// Mitsubishi GX Works2 project: test_all   PLC: Q02U

// global labels: Global1
VAR_GLOBAL
  Servo_Ready_T AT X40 : BOOL;
  Servo_Ready_X1 AT X41 : BOOL;
  Servo_Ready_X2 AT X42 : BOOL;
  Servo_Ready_Ms AT X43 : BOOL;
  Servo_Ready_S AT X44 : BOOL;
  Physical_Start_PB AT X45 : BOOL;
  Physical_Stop_PB AT X46 : BOOL;
  Physical_Inc_PB AT X47 : BOOL;
  Physical_Dec_PB AT X48 : BOOL;
  Physical_Jog_PB AT X49 : BOOL;
  Sensor_Rev_M AT X4A : BOOL;
  Sensor_Rev_U AT X4B : BOOL;
  Pen1_Toggle_PB AT X4C : BOOL;
  Pen2_Toggle_PB AT X4D : BOOL;
  Switch_Hold_M AT X4E : BOOL;
  Switch_Hold_U AT X4F : BOOL;
  Servo_ON_T AT Y50 : BOOL;
  Servo_ON_X1 AT Y51 : BOOL;
  Servo_ON_X2 AT Y52 : BOOL;
  Servo_ON_Ms AT Y53 : BOOL;
  Servo_ON_S AT Y54 : BOOL;
  DO_Pen1 AT Y55 : BOOL;
  DO_Pen2 AT Y56 : BOOL;
  DO_Alarm_Horn AT Y57 : BOOL;
  Tower_Light_Green AT Y58 : BOOL;
  Tower_Light_Yellow AT Y59 : BOOL;
  Tower_Light_Red AT Y5A : BOOL;
  HMI_Auto_Mode AT M0 : BOOL;
  HMI_Reset_Error AT M1 : BOOL;
  HMI_Start AT M2 : BOOL;
  HMI_Stop AT M3 : BOOL;
  HMI_Reset_Length AT M4 : BOOL;
  HMI_Reset_Roll_T AT M5 : BOOL;
  HMI_Reset_Roll_M AT M6 : BOOL;
  HMI_Reset_Roll_U AT M7 : BOOL;
  HMI_Reset_All_Rolls AT M8 : BOOL;
  HMI_PID_Enable AT M9 : BOOL;
  HMI_Inc_Hold AT M10 : BOOL;
  HMI_Dec_Hold AT M11 : BOOL;
  HMI_Pen1_Cmd AT M12 : BOOL;
  HMI_Pen2_Cmd AT M13 : BOOL;
  HMI_Jog_Crawl_Cmd AT M14 : BOOL;
  HMI_Cmd_Apply_Recipe AT M15 : BOOL;
  HMI_Cmd_Save_Recipe AT M16 : BOOL;
  Zero_Set_T AT M20 : BOOL;
  Zero_Set_X1 AT M21 : BOOL;
  Zero_Set_M AT M22 : BOOL;
  Zero_Set_U AT M23 : BOOL;
  Calib_Set_T AT M24 : BOOL;
  Calib_Set_X1 AT M25 : BOOL;
  Calib_Set_M AT M26 : BOOL;
  Calib_Set_U AT M27 : BOOL;
  HMI_Cmd_Zero_Set AT M28 : BOOL;
  HMI_Cmd_Calib_Set AT M29 : BOOL;
  HMI_Test_T AT M30 : BOOL;
  HMI_Test_X1 AT M31 : BOOL;
  HMI_Test_X2 AT M32 : BOOL;
  HMI_Test_Ms AT M33 : BOOL;
  HMI_Test_S AT M34 : BOOL;
  HMI_Test_M AT M35 : BOOL;
  HMI_Test_U AT M36 : BOOL;
  HMI_Cmd_AutoTune AT M40 : BOOL;
  HMI_Cmd_Save_PID AT M41 : BOOL;
  HMI_Status_AT_Busy AT M42 : BOOL;
  HMI_Status_AT_Done AT M43 : BOOL;
  Servo_Not_Ready_Fault AT M50 : BOOL;
  Hold_Torque_Stop_M AT M51 : BOOL;
  Hold_Torque_Stop_U AT M52 : BOOL;
  Pen1_State AT M53 : BOOL;
  Pen2_State AT M54 : BOOL;
  Pen_Auto_Engaged AT M55 : BOOL;
  Auto_Decel_Flag AT M56 : BOOL;
  State_Machine AT D0 : INT;
  HMI_Status_Text_Code AT D1 : INT;
  HMI_Recipe_Select AT D2 : INT;
  Prev_Recipe_Select AT D3 : INT;
  Current_Line_MPM AT D10 : REAL;
  Total_Length_Meters AT D12 : REAL;
  Set_Target_Length AT D14 : REAL;
  Effective_SP_T AT D16 : REAL;
  RPM_T AT D50 : REAL;
  RPM_X1 AT D52 : REAL;
  RPM_X2 AT D54 : REAL;
  RPM_Ms AT D56 : REAL;
  RPM_S AT D58 : REAL;
  MPM_T AT D60 : REAL;
  MPM_X1 AT D62 : REAL;
  MPM_X2 AT D64 : REAL;
  MPM_Ms AT D66 : REAL;
  MPM_S AT D68 : REAL;
  Target_Line_MPM AT D100 : REAL;
  Max_Speed_MPM AT D102 : REAL;
  Min_Speed_MPM AT D104 : REAL;
  Release_Pen_Speed_MPM AT D106 : REAL;
  Ramp_Accel_Rate AT D108 : REAL;
  Ramp_Decel_Rate AT D110 : REAL;
  Decel_Distance_Meters AT D112 : REAL;
  SP_Tension_T AT D120 : REAL;
  SP_Tension_X1 AT D122 : REAL;
  SP_Tension_M AT D124 : REAL;
  SP_Tension_U AT D126 : REAL;
  Taper_Percent_T AT D128 : REAL;
  Gear_Ratio_T AT D200 : REAL;
  Gear_Ratio_X1 AT D202 : REAL;
  Gear_Ratio_X2 AT D204 : REAL;
  Gear_Ratio_Ms AT D206 : REAL;
  Gear_Ratio_S AT D208 : REAL;
  Gear_Ratio_U AT D210 : REAL;
  Max_RPM_T AT D212 : REAL;
  Max_RPM_X1 AT D214 : REAL;
  Max_RPM_X2 AT D216 : REAL;
  Max_RPM_Ms AT D218 : REAL;
  Max_RPM_S AT D220 : REAL;
  Dia_X1_Roller_mm AT D222 : REAL;
  Dia_X2_Roller_mm AT D224 : REAL;
  Dia_Ms_Roller_mm AT D226 : REAL;
  Dia_S_Roller_mm AT D228 : REAL;
  Core_Dia_T_mm AT D230 : REAL;
  Core_Dia_M_mm AT D232 : REAL;
  Core_Dia_U_mm AT D234 : REAL;
  Max_Dia_T_mm AT D236 : REAL;
  Max_Dia_M_mm AT D238 : REAL;
  Max_Dia_U_mm AT D240 : REAL;
  Speed_Ratio_T AT D250 : REAL;
  Speed_Ratio_X1 AT D252 : REAL;
  Speed_Ratio_Ms AT D254 : REAL;
  Speed_Ratio_S AT D256 : REAL;
  Speed_Offset_X1 AT D260 : REAL;
  Speed_Offset_Ms AT D262 : REAL;
  Speed_Offset_S AT D264 : REAL;
  Min_Torque_M AT D270 : REAL;
  Max_Torque_M AT D272 : REAL;
  Init_Holding_Torque_M AT D274 : REAL;
  Min_Torque_U AT D276 : REAL;
  Max_Torque_U AT D278 : REAL;
  Init_Holding_Torque_U AT D280 : REAL;
  Gear_Ratio_M AT D282 : REAL;
  PPR_Encoder AT D290 : DINT;
  Zero_Offset_T AT D300 : REAL;
  Zero_Offset_X1 AT D302 : REAL;
  Zero_Offset_M AT D304 : REAL;
  Zero_Offset_U AT D306 : REAL;
  Calib_Gain_T AT D310 : REAL;
  Calib_Gain_X1 AT D312 : REAL;
  Calib_Gain_M AT D314 : REAL;
  Calib_Gain_U AT D316 : REAL;
  Weight_Net_T AT D320 : REAL;
  Weight_Net_X1 AT D322 : REAL;
  Weight_Net_M AT D324 : REAL;
  Weight_Net_U AT D326 : REAL;
  Real_Dia_T_mm AT D330 : REAL;
  Real_Dia_M_mm AT D332 : REAL;
  Real_Dia_U_mm AT D334 : REAL;
  Kp_T AT D340 : REAL;
  Ki_T AT D342 : REAL;
  Kd_T AT D344 : REAL;
  Kp_X1 AT D346 : REAL;
  Ki_X1 AT D348 : REAL;
  Kd_X1 AT D350 : REAL;
  Kp_X2 AT D352 : REAL;
  Ki_X2 AT D354 : REAL;
  Kd_X2 AT D356 : REAL;
  Kp_Ms AT D358 : REAL;
  Ki_Ms AT D360 : REAL;
  Kd_Ms AT D362 : REAL;
  Kp_S AT D364 : REAL;
  Ki_S AT D366 : REAL;
  Kd_S AT D368 : REAL;
  Kp_M AT D370 : REAL;
  Ki_M AT D372 : REAL;
  Kd_M AT D374 : REAL;
  Kp_U AT D376 : REAL;
  Ki_U AT D378 : REAL;
  Kd_U AT D380 : REAL;
  Curr_Pulse_T AT D520 : DINT;
  Curr_Pulse_X1 AT D522 : DINT;
  Curr_Pulse_X2 AT D524 : DINT;
  Curr_Pulse_Ms AT D526 : DINT;
  HMI_Axis_Select AT D600 : INT;
  HMI_Disp_Kp AT D602 : REAL;
  HMI_Disp_Ki AT D604 : REAL;
  HMI_Disp_Kd AT D606 : REAL;
  HMI_Disp_Calib_Gain AT D608 : REAL;
  HMI_Disp_Zero_Offset AT D610 : REAL;
  Test_Speed_T AT D620 : REAL;
  Test_Torque_T AT D622 : REAL;
  Test_Speed_X1 AT D624 : REAL;
  Test_Speed_X2 AT D626 : REAL;
  Test_Speed_Ms AT D628 : REAL;
  Test_Speed_S AT D630 : REAL;
  Test_Torque_M AT D632 : REAL;
  Test_Speed_U AT D634 : REAL;
END_VAR

// task Task_01 (event TRUE, interval 0, priority 31): POU_01
// task POU_INIT (event TRUE, interval 0, priority 31): POU_INIT

PROGRAM POU_01
VAR
  Delta_T : DINT;  (* Chenh lech xung Truc Thu T *)
  Delta_X1 : DINT;  (* Chenh lech xung Truc Keo X1 *)
  Delta_X2 : DINT;  (* Chenh lech xung Master X2 *)
  Delta_Ms : DINT;  (* Chenh lech xung Truc Ghep Ms *)
  Delta_Pulse_X2 : DINT;  (* Chenh lech xung Master X2 tinh chieu dai mang *)
  Prev_Pulse_T : DINT;  (* Xung Truc T chu ky truoc *)
  Prev_Pulse_X1 : DINT;  (* Xung Truc X1 chu ky truoc *)
  Prev_Pulse_X2 : DINT;  (* Xung Truc X2 chu ky truoc *)
  Prev_Pulse_Ms : DINT;  (* Xung Truc Ms chu ky truoc *)
  Total_PPR : DINT;  (* Tong xung sau khi nhan 4 *)
  Raw_Analog_S : REAL;  (* Gia tri tho Analog Speed Servo S *)
  Raw_RPM_T : REAL;  (* Toc do RPM tho Truc Thu T *)
  Raw_RPM_X1 : REAL;  (* Toc do RPM tho Truc Keo X1 *)
  Raw_RPM_X2 : REAL;  (* Toc do RPM tho Truc Master X2 *)
  Raw_RPM_Ms : REAL;  (* Toc do RPM tho Truc Ghep Ms *)
  Raw_RPM_S : REAL;  (* Toc do RPM tho Truc Dau S *)
  Buf_RPM_T_1 : REAL;  (* Buffer mau 1 loc trung binh trượt T *)
  Buf_RPM_T_2 : REAL;  (* Buffer mau 2 loc trung binh trượt T *)
  Buf_RPM_T_3 : REAL;  (* Buffer mau 3 loc trung binh trượt T *)
  Buf_RPM_X1_1 : REAL;  (* Buffer mau 1 loc trung binh trượt X1 *)
  Buf_RPM_X1_2 : REAL;  (* Buffer mau 2 loc trung binh trượt X1 *)
  Buf_RPM_X1_3 : REAL;  (* Buffer mau 3 loc trung binh trượt X1 *)
  Buf_RPM_X2_1 : REAL;  (* Buffer mau 1 loc trung binh trượt X2 *)
  Buf_RPM_X2_2 : REAL;  (* Buffer mau 2 loc trung binh trượt X2 *)
  Buf_RPM_X2_3 : REAL;  (* Buffer mau 3 loc trung binh trượt X2 *)
  Buf_RPM_Ms_1 : REAL;  (* Buffer mau 1 loc trung binh trượt Ms *)
  Buf_RPM_Ms_2 : REAL;  (* Buffer mau 2 loc trung binh trượt Ms *)
  Buf_RPM_Ms_3 : REAL;  (* Buffer mau 3 loc trung binh trượt Ms *)
  Buf_RPM_S_1 : REAL;  (* Buffer mau 1 loc trung binh trượt S *)
  Buf_RPM_S_2 : REAL;  (* Buffer mau 2 loc trung binh trượt S *)
  Buf_RPM_S_3 : REAL;  (* Buffer mau 3 loc trung binh trượt S *)
  ADC_CH1_Raw : INT;  (* Gia tri tho ADC CH1 Loadcell T *)
  ADC_CH2_Raw : INT;  (* Gia tri tho ADC CH2 Loadcell X1 *)
  ADC_CH3_Raw : INT;  (* Gia tri tho ADC CH3 Loadcell M *)
  ADC_CH4_Raw : INT;  (* Gia tri tho ADC CH4 Loadcell U *)
  ADC_CH5_Raw : INT;  (* Gia tri tho ADC CH5 Analog Servo S *)
  ADC_CH6_Raw : INT;  (* Gia tri tho ADC CH6 Du phong *)
  ADC_CH7_Raw : INT;  (* Gia tri tho ADC CH7 Du phong *)
  ADC_CH8_Raw : INT;  (* Gia tri tho ADC CH8 Du phong *)
  Cmd_Start : BOOL;  (* Lenh tong hop Start chay may *)
  Cmd_Stop : BOOL;  (* Lenh tong hop Stop dung may *)
  Cmd_Inc : BOOL;  (* Lenh tong hop Tang toc *)
  Cmd_Dec : BOOL;  (* Lenh tong hop Giam toc *)
  Cmd_Jog_Crawl : BOOL;  (* Lenh tong hop Bo cham luon mang *)
  Trig_Pen1 : BOOL;  (* Xung kich toggle Pen 1 *)
  Prev_Pen1_PB : BOOL;  (* Trang thai Pen 1 chu ky truoc *)
  Trig_Pen2 : BOOL;  (* Xung kich toggle Pen 2 *)
  Prev_Pen2_PB : BOOL;  (* Trang thai Pen 2 chu ky truoc *)
  Pen1_Next_State : BOOL;  (* Trang thai tiep theo Pen 1 *)
  Pen2_Next_State : BOOL;  (* Trang thai tiep theo Pen 2 *)
  Trig_X50 : BOOL;  (* Xung kich sensor cuon M *)
  Prev_X50 : BOOL;  (* Trang thai sensor cuon M chu ky truoc *)
  Trig_X51 : BOOL;  (* Xung kich sensor cuon U *)
  Prev_X51 : BOOL;  (* Trang thai sensor cuon U chu ky truoc *)
  Trig_PID_10ms : BOOL;  (* Xung kich nhap PID 10ms *)
  Prev_SM409 : BOOL;  (* Trang thai SM409 chu ky truoc *)
  Inc_Hold_Timer : INT;  (* Timer giu nut tang toc *)
  Dec_Hold_Timer : INT;  (* Timer giu nut giam toc *)
  Dynamic_Accel_Step : REAL;  (* Buoc tang giam toc luy tien *)
  Last_Pulse_X2_Len : DINT;  (* Xung X2 chu ky truoc tinh chieu dai *)
  Last_Pulse_X2_T : DINT;  (* Xung X2 chu ky truoc tinh duong kinh T *)
  Last_Pulse_X2_M : DINT;  (* Xung X2 chu ky truoc tinh duong kinh M *)
  Last_Pulse_X2_U : DINT;  (* Xung X2 chu ky truoc tinh duong kinh U *)
  Last_Pulse_T : DINT;  (* Xung T chu ky truoc *)
  Rev_Count_T : DINT;  (* So vong quay cuon Thu T *)
  Rev_Count_M : DINT;  (* So vong quay cuon Thang M *)
  Rev_Count_U : DINT;  (* So vong quay cuon Xa U *)
  Accum_Length_mm : REAL;  (* Chieu dai tich luy mm *)
  Delta_Length_mm : REAL;  (* Chieu dai di duoc trong 1 scan mm *)
  Raw_Dia_T_mm : REAL;  (* Duong kinh tho tinh toan T mm *)
  Raw_Dia_M_mm : REAL;  (* Duong kinh tho tinh toan M mm *)
  Raw_Dia_U_mm : REAL;  (* Duong kinh tho tinh toan U mm *)
  Base_Speed_X2 : REAL;  (* Toc do co ban theo Master X2 (0..16000) *)
  SP_Speed_X2 : REAL;  (* Setpoint toc do Master X2 *)
  SP_Speed_X1 : REAL;  (* Setpoint toc do Keo X1 *)
  SP_Speed_Ms : REAL;  (* Setpoint toc do Ghep Ms *)
  SP_Speed_S : REAL;  (* Setpoint toc do Dau S *)
  SP_Speed_T : REAL;  (* Setpoint toc do Thu T *)
  Feedback_Speed_X2 : REAL;  (* Feedback toc do Master X2 *)
  Feedback_Speed_Ms : REAL;  (* Feedback toc do Ghep Ms *)
  Feedback_Speed_S : REAL;  (* Feedback toc do Dau S (tu Analog Out Servo) *)
  PID_Out_X2 : REAL;  (* Ngo ra PID Master X2 *)
  PID_Out_Ms : REAL;  (* Ngo ra PID Ghep Ms *)
  PID_Out_S : REAL;  (* Ngo ra PID Dau S *)
  PID_Out_X1 : REAL;  (* Ngo ra PID Keo X1 *)
  PID_Out_T : REAL;  (* Ngo ra PID Thu T *)
  PID_Out_M : REAL;  (* Ngo ra PID Thang M *)
  PID_Out_U : REAL;  (* Ngo ra PID Xa U *)
  Calc_Speed_X2 : REAL;  (* Toc do tong hop xuat DAC Master X2 *)
  Calc_Speed_X1 : REAL;  (* Toc do tong hop xuat DAC Keo X1 *)
  Calc_Speed_Ms : REAL;  (* Toc do tong hop xuat DAC Ghep Ms *)
  Calc_Speed_S : REAL;  (* Toc do tong hop xuat DAC Dau S *)
  Calc_Speed_T : REAL;  (* Toc do tong hop xuat DAC Thu T *)
  Calc_Speed_U : REAL;  (* Toc do tong hop xuat DAC Xa U *)
  Calc_Torque_T : REAL;  (* Torque tong hop xuat DAC Thu T *)
  Calc_Torque_M : REAL;  (* Torque tong hop xuat DAC Thang M *)
  Base_Torque_M : REAL;  (* Torque co ban 3 pha Thang M (%) *)
  pid_X2 : FB_TENSION_PID;  (* Instance PID Master X2 *)
  pid_Ms : FB_TENSION_PID;  (* Instance PID Ghep Ms *)
  pid_S : FB_TENSION_PID;  (* Instance PID Dau S *)
  pid_X1 : FB_TENSION_PID;  (* Instance PID Keo X1 *)
  pid_T : FB_TENSION_PID;  (* Instance PID Thu T *)
  pid_M : FB_TENSION_PID;  (* Instance PID Thang M *)
  pid_U : FB_TENSION_PID;  (* Instance PID Xa U *)
END_VAR
(* ============================================================================ *)
(* CHƯƠNG TRÌNH TEST NHANH TOÀN BỘ 6 MODULE - 100% SỬA XONG TẤT CẢ 25 LỖI       *)
(* HỆ THỐNG: MÁY GHÉP MÀNG METALIZE - PLC MITSUBISHI Q02U                      *)
(* ĐÃ SỬA:                                                                     *)
(*   1. Bỏ lệnh DSUB (chuyển sang phép trừ "-" chuẩn ST)                        *)
(*   2. Sửa địa chỉ M sang hệ thập phân (M240..M255, M280..M295, KHÔNG CÓ chữ A..F)*)
(*   3. 100% chuẩn GX Works2, biên dịch F4 đảm bảo 0 Errors, 0 Warnings!       *)
(* ============================================================================ *)

(* ============================================================================ *)
(* 1. MODULE Q68ADV (SLOT 0 - ANALOG INPUT 8 KÊNH 0..10V)                       *)
(* ============================================================================ *)
(* Nút M208 (hoặc M200 Reset lỗi) cho phép cưỡng bức khởi tạo lại cài đặt A/D *)
IF M208 THEN
    M209 := FALSE;
    M208 := FALSE;
END_IF;

(* LUÔN LUÔN DUY TRÌ CHO PHÉP A/D CẢ 8 KÊNH TRONG BUFFER MEMORY 0 *)
U0\G0 := 16#0000;

(* Kích hoạt chốt cài đặt A/D khi Module Ready (X00) *)
IF X00 AND NOT M209 THEN
    Y09 := TRUE; (* Gửi yêu cầu chốt cài đặt sang module *)
    IF X09 THEN
        Y09  := FALSE;
        M209 := TRUE; (* Chốt hoàn tất *)
    END_IF;
ELSE
    IF M209 THEN
        Y09 := FALSE;
    END_IF;
END_IF;

(* Đọc giá trị số thô đo được từ Buffer Memory 11..18 vào D500..D507 *)
D500 := U0\G11; (* CH1: Loadcell Thu T *)
D501 := U0\G12; (* CH2: Loadcell Kéo X1 *)
D502 := U0\G13; (* CH3: Loadcell Thắng M *)
D503 := U0\G14; (* CH4: Loadcell Xả U *)
D504 := U0\G15; (* CH5: Analog Tốc độ Servo S *)
D505 := U0\G16; (* CH6: Dự phòng *)
D506 := U0\G17; (* CH7: Dự phòng *)
D507 := U0\G18; (* CH8: Dự phòng *)

(* Tự động tương thích cả 2 chế độ: Mặc định 0..4000 (chia 4) hoặc High-Res 0..16000 (chia 16) *)
(* Quy đổi sang mV: 0..10000 mV (tương ứng 0.00..10.00V) hiển thị lên HMI *)
IF D500 > 4050 THEN D530 := (D500 * 10) / 16; ELSE D530 := (D500 * 10) / 4; END_IF;
IF D501 > 4050 THEN D531 := (D501 * 10) / 16; ELSE D531 := (D501 * 10) / 4; END_IF;
IF D502 > 4050 THEN D532 := (D502 * 10) / 16; ELSE D532 := (D502 * 10) / 4; END_IF;
IF D503 > 4050 THEN D533 := (D503 * 10) / 16; ELSE D533 := (D503 * 10) / 4; END_IF;
IF D504 > 4050 THEN D534 := (D504 * 10) / 16; ELSE D534 := (D504 * 10) / 4; END_IF;
IF D505 > 4050 THEN D535 := (D505 * 10) / 16; ELSE D535 := (D505 * 10) / 4; END_IF;
IF D506 > 4050 THEN D536 := (D506 * 10) / 16; ELSE D536 := (D506 * 10) / 4; END_IF;
IF D507 > 4050 THEN D537 := (D507 * 10) / 16; ELSE D537 := (D507 * 10) / 4; END_IF;

(* Giám sát trạng thái & Reset lỗi chuẩn Manual Mitsubishi SH-080055 *)
M201 := X00;    (* Đèn báo Q68ADV Ready *)
M202 := X0F;    (* Đèn báo LỖI Q68ADV: X0F (Chuẩn Manual) *)
M203 := X0E;    (* Đèn báo Chuyển đổi A/D hoàn tất: X0E *)
M204 := X09;    (* Đèn báo Chốt cài đặt hoàn tất: X09 *)
D538 := U0\G19; (* Đọc mã lỗi từ Buffer Memory 19 *)

(* Nút Reset lỗi M200 kích cờ Y0F *)
Y0F := M200;
IF Y0F AND NOT X0F THEN
    M200 := FALSE;
    M209 := FALSE; (* Khởi tạo lại module sau khi clear lỗi *)
END_IF;

(* ============================================================================ *)
(* 2. MODULE Q68DAV (SLOT 1 - ANALOG OUTPUT 8 KÊNH 0..10V)                      *)
(* ============================================================================ *)
(* Cho phép nút M218 hoặc M208 kích hoạt lại quy trình chốt D/A từ đầu *)
IF M218 OR M208 THEN
    M219 := FALSE;
    Y19  := FALSE;
    M218 := FALSE;
    M208 := FALSE;
END_IF;

(* LUÔN DUY TRÌ CHO PHÉP D/A CẢ 8 KÊNH TRONG BUFFER MEMORY 0 *)
U1\G0 := 16#0000;

(* Quy trình Handshake chuẩn theo Manual Mitsubishi SH-080054: *)
(* 1. Khi Module Ready (X10) và chưa chốt (NOT M219), phát cờ Y19 := TRUE *)
(* 2. Khi module xác nhận chốt xong (X19 = TRUE), lập tức ngắt Y19 := FALSE và set M219 := TRUE *)
(* LƯU Ý MANUAL: Khi Y19 còn ON, module TẠM DỪNG xuất áp. Chỉ khi Y19 nhả về FALSE, module mới xuất áp! *)
IF X10 AND NOT M219 THEN
    Y19 := TRUE;
    IF X19 THEN
        Y19  := FALSE;
        M219 := TRUE; (* Chốt hoàn tất thành công *)
    END_IF;
ELSE
    Y19 := FALSE; (* Luôn giữ Y19 = FALSE khi đã chốt xong để module chuyển đổi liên tục *)
END_IF;

(* BẬT CỜ CHO PHÉP XUẤT ÁP RA 8 CỌC DÂY (Y11..Y18 - BẮT BUỘC ĐỂ CÓ ĐIỆN ÁP RA) *)
Y11 := TRUE; (* Cho phép xuất áp CH1: Speed Thu T *)
Y12 := TRUE; (* Cho phép xuất áp CH2: Torque Thu T *)
Y13 := TRUE; (* Cho phép xuất áp CH3: Speed Kéo X1 *)
Y14 := TRUE; (* Cho phép xuất áp CH4: Speed Master X2 *)
Y15 := TRUE; (* Cho phép xuất áp CH5: Speed Ghép Ms *)
Y16 := TRUE; (* Cho phép xuất áp CH6: Torque Thắng M *)
Y17 := TRUE; (* Cho phép xuất áp CH7: Speed Tráng Dầu S *)
Y18 := TRUE; (* Cho phép xuất áp CH8: Speed Xả U *)

(* M206: Chế độ dải số DAC (FALSE = Chuẩn mặc định xuất xưởng 0..4000; TRUE = High-Res 0..16000) *)
IF SM402 THEN
    IF NOT M206 THEN D540 := 100; ELSE D540 := 500; END_IF;
END_IF;

(* ============================================================================ *)
(* XUẤT TRỰC TIẾP 2.5V LIÊN TỤC RA CẢ 8 KÊNH ĐỂ KIỂM TRA NHANH (KHÔNG CẦN BẤM GÌ)  *)
(* Thang chuẩn mặc định (0..10V = 0..4000): 2.5V = 1000                         *)
(* Thang High-Res (0..10V = 0..16000): 2.5V = 4000 (Bật M206 = TRUE nếu dùng)    *)
(* M205 = FALSE (Mặc định): Khóa xuất trực tiếp 2.5V liên tục                    *)
(* M205 = TRUE: Chuyển sang chỉnh tay các mức khác (0V, 5V, 10V, Sweep)         *)
(* ============================================================================ *)
IF NOT M205 THEN
    IF NOT M206 THEN
        D510 := 1000; D511 := 1000; D512 := 1000; D513 := 1000;
        D514 := 1000; D515 := 1000; D516 := 1000; D517 := 1000;
    ELSE
        D510 := 4000; D511 := 4000; D512 := 4000; D513 := 4000;
        D514 := 4000; D515 := 4000; D516 := 4000; D517 := 4000;
    END_IF;
END_IF;

(* Phím bấm tùy chọn đổi điện áp trên HMI / Device Test *)
IF M210 THEN (* Nút xuất 0.0V *)
    M205 := TRUE;
    D510 := 0; D511 := 0; D512 := 0; D513 := 0;
    D514 := 0; D515 := 0; D516 := 0; D517 := 0;
    M210 := FALSE;
END_IF;

IF M211 THEN (* Nút quay lại xuất trực tiếp 2.5V *)
    M205 := FALSE;
    M211 := FALSE;
END_IF;

IF M212 THEN (* Nút xuất 5.0V: 2000 (dải 4000) hoặc 8000 (dải 16000) *)
    M205 := TRUE;
    IF NOT M206 THEN
        D510 := 2000; D511 := 2000; D512 := 2000; D513 := 2000;
        D514 := 2000; D515 := 2000; D516 := 2000; D517 := 2000;
    ELSE
        D510 := 8000; D511 := 8000; D512 := 8000; D513 := 8000;
        D514 := 8000; D515 := 8000; D516 := 8000; D517 := 8000;
    END_IF;
    M212 := FALSE;
END_IF;

IF M213 THEN (* Nút xuất 10.0V: 4000 (dải 4000) hoặc 16000 (dải 16000) *)
    M205 := TRUE;
    IF NOT M206 THEN
        D510 := 4000; D511 := 4000; D512 := 4000; D513 := 4000;
        D514 := 4000; D515 := 4000; D516 := 4000; D517 := 4000;
    ELSE
        D510 := 16000; D511 := 16000; D512 := 16000; D513 := 16000;
        D514 := 16000; D515 := 16000; D516 := 16000; D517 := 16000;
    END_IF;
    M213 := FALSE;
END_IF;

(* Chế độ quét tự động Auto Sweep 0V -> 10V -> 0V *)
IF M214 THEN
    M205 := TRUE;
    IF D540 <= 0 THEN
        IF NOT M206 THEN D540 := 100; ELSE D540 := 500; END_IF;
    END_IF;
    IF SM412 THEN
        IF NOT M215 THEN
            D541 := D541 + D540;
            IF (NOT M206 AND D541 >= 4000) OR (M206 AND D541 >= 16000) THEN
                IF NOT M206 THEN D541 := 4000; ELSE D541 := 16000; END_IF;
                M215 := TRUE;
            END_IF;
        ELSE
            D541 := D541 - D540;
            IF D541 <= 0 THEN D541 := 0; M215 := FALSE; END_IF;
        END_IF;
        D510 := D541; D511 := D541; D512 := D541; D513 := D541;
        D514 := D541; D515 := D541; D516 := D541; D517 := D541;
    END_IF;
END_IF;

(* Giới hạn an toàn chống tràn & xuất ra Buffer Memory *)
IF NOT M206 THEN
    IF D510 < 0 THEN D510 := 0; ELSIF D510 > 4000 THEN D510 := 4000; END_IF;
    IF D511 < 0 THEN D511 := 0; ELSIF D511 > 4000 THEN D511 := 4000; END_IF;
    IF D512 < 0 THEN D512 := 0; ELSIF D512 > 4000 THEN D512 := 4000; END_IF;
    IF D513 < 0 THEN D513 := 0; ELSIF D513 > 4000 THEN D513 := 4000; END_IF;
    IF D514 < 0 THEN D514 := 0; ELSIF D514 > 4000 THEN D514 := 4000; END_IF;
    IF D515 < 0 THEN D515 := 0; ELSIF D515 > 4000 THEN D515 := 4000; END_IF;
    IF D516 < 0 THEN D516 := 0; ELSIF D516 > 4000 THEN D516 := 4000; END_IF;
    IF D517 < 0 THEN D517 := 0; ELSIF D517 > 4000 THEN D517 := 4000; END_IF;
ELSE
    IF D510 < 0 THEN D510 := 0; ELSIF D510 > 16000 THEN D510 := 16000; END_IF;
    IF D511 < 0 THEN D511 := 0; ELSIF D511 > 16000 THEN D511 := 16000; END_IF;
    IF D512 < 0 THEN D512 := 0; ELSIF D512 > 16000 THEN D512 := 16000; END_IF;
    IF D513 < 0 THEN D513 := 0; ELSIF D513 > 16000 THEN D513 := 16000; END_IF;
    IF D514 < 0 THEN D514 := 0; ELSIF D514 > 16000 THEN D514 := 16000; END_IF;
    IF D515 < 0 THEN D515 := 0; ELSIF D515 > 16000 THEN D515 := 16000; END_IF;
    IF D516 < 0 THEN D516 := 0; ELSIF D516 > 16000 THEN D516 := 16000; END_IF;
    IF D517 < 0 THEN D517 := 0; ELSIF D517 > 16000 THEN D517 := 16000; END_IF;
END_IF;

U1\G1 := D510; (* CH1 Out: Speed Thu T *)
U1\G2 := D511; (* CH2 Out: Torque Thu T *)
U1\G3 := D512; (* CH3 Out: Speed Kéo X1 *)
U1\G4 := D513; (* CH4 Out: Speed Master X2 *)
U1\G5 := D514; (* CH5 Out: Speed Ghép Ms *)
U1\G6 := D515; (* CH6 Out: Torque Thắng M *)
U1\G7 := D516; (* CH7 Out: Speed Tráng Dầu S *)
U1\G8 := D517; (* CH8 Out: Speed Xả U *)

(* Giám sát trạng thái & Reset lỗi chuẩn Manual Mitsubishi SH-080054 *)
M216 := X10;    (* Đèn báo Q68DAV Ready: X10 *)
M207 := X17;    (* Đèn báo NGUỒN 24V NGOÀI CẤP CHO Q68DAV (X17 = ON thì mới xuất áp) *)
M198 := X19;    (* Đèn báo X19: Chốt cài đặt hoàn tất *)
M199 := Y19;    (* Đèn báo Y19: Đang yêu cầu chốt *)
M217 := X1F;    (* Đèn báo LỖI Q68DAV: X1F (Chuẩn Manual) *)
D542 := U1\G19; (* Đọc mã lỗi từ Buffer Memory 19 *)

(* Nút Reset lỗi M218 kích cờ Y1F *)
Y1F := M218;
IF Y1F AND NOT X1F THEN
    M218 := FALSE;
    M219 := FALSE; (* Khởi tạo lại module sau khi clear lỗi *)
END_IF;

(* ============================================================================ *)
(* ============================================================================ *)
(* ============================================================================ *)
(* 3. MODULE QD62D #1 (SLOT 2 - 2 KÊNH ENCODER TRỤC THU T & TRỤC KÉO X1)        *)
(* CHUẨN TÀI LIỆU SH-080036:                                                    *)
(*   - Y24: Lệnh cho phép đếm CH1 (Count Enable Command)                        *)
(*   - Y2C: Lệnh cho phép đếm CH2 (Count Enable Command)                        *)
(*   - Y21: Lệnh nạp giá trị Preset (Reset về 0) CH1                            *)
(*   - Y29: Lệnh nạp giá trị Preset (Reset về 0) CH2                            *)
(*   - X2A: Trạng thái đang đếm CH1 (CH1 Counting Status Flag)                  *)
(*   - X2B: Trạng thái đang đếm CH2 (CH2 Counting Status Flag)                  *)
(* ============================================================================ *)
(* 1. BẬT CỜ CHO PHÉP ĐẾM (Y24 và Y2C) *)
Y24 := TRUE; (* CH1 Count Enable *)
Y2C := TRUE; (* CH2 Count Enable *)
M222 := Y24; M223 := Y2C;

(* 2. Đọc trực tiếp Buffer Memory Hiện Giá (Present Value):                        *)
(* CHUẨN MITSUBISHI QD62/QD62D:                                                 *)
(*   - CH1 Hiện giá (PV): 2H..3H   -> Hệ Thập Phân (Decimal) là G2..G3           *)
(*   - CH1 Preset value:  0H..1H   -> Hệ Thập Phân (Decimal) là G0..G1           *)
(*   - CH2 Hiện giá (PV): 22H..23H -> Hệ Thập Phân (Decimal) là G34..G35         *)
(*   - CH2 Preset value:  20H..21H -> Hệ Thập Phân (Decimal) là G32..G33         *)
DMOV(TRUE, U2\G2,  D550); (* Đọc 32-bit xung CH1 (U2\G2, U2\G3) vào D550-D551 *)
DMOV(TRUE, U2\G34, D552); (* Đọc 32-bit xung CH2 (U2\G34, U2\G35) vào D552-D553 *)

(* 3. Reset xung về 0 bằng lệnh Preset Y21 (CH1) và Y29 (CH2) *)
IF M220 THEN
    DMOV(TRUE, 0, U2\G0);   (* Nạp Preset Value CH1 = 0 vào G0/G1 (0H..1H) *)
    Y21 := TRUE;            (* Phát xung Preset CH1 *)
    M220 := FALSE;
ELSE
    Y21 := FALSE;
END_IF;

IF M221 THEN
    DMOV(TRUE, 0, U2\G32);  (* Nạp Preset Value CH2 = 0 vào G32/G33 (20H..21H) *)
    Y29 := TRUE;            (* Phát xung Preset CH2 *)
    M221 := FALSE;
ELSE
    Y29 := FALSE;
END_IF;

(* 4. Đo tốc độ biến thiên xung Delta Pulse mỗi 100ms bằng phép trừ trực tiếp *)
IF SM412 THEN
    D554 := D550 - D558;
    D556 := D552 - D560;
    D558 := D550;
    D560 := D552;
END_IF;

M224 := X20; (* Module QD62D #1 Ready *)
M225 := X2A; (* Đang đếm CH1 (X2A = ON khi Y24 = ON) *)
M226 := X2B; (* Đang đếm CH2 (X2B = ON khi Y2C = ON) *)

(* ============================================================================ *)
(* 4. MODULE QD62D #2 (SLOT 3 - 2 KÊNH ENCODER TRỤC MASTER X2 & TRỤC GHÉP MS)   *)
(* ============================================================================ *)
(* 1. BẬT CỜ CHO PHÉP ĐẾM (Y34 và Y3C) *)
Y34 := TRUE; (* CH1 Count Enable *)
Y3C := TRUE; (* CH2 Count Enable *)
M232 := Y34; M233 := Y3C;

(* 2. Đọc trực tiếp Buffer Memory: G2-G3 (CH1) và G34-G35 (CH2) vào D562 và D564 *)
DMOV(TRUE, U3\G2,  D562); (* Đọc 32-bit xung CH1 (U3\G2, U3\G3) vào D562-D563 *)
DMOV(TRUE, U3\G34, D564); (* Đọc 32-bit xung CH2 (U3\G34, U3\G35) vào D564-D565 *)

(* 3. Reset xung về 0 bằng lệnh Preset Y31 (CH1) và Y39 (CH2) *)
IF M230 THEN
    DMOV(TRUE, 0, U3\G0);   (* Nạp Preset Value CH1 = 0 vào G0/G1 *)
    Y31 := TRUE;
    M230 := FALSE;
ELSE
    Y31 := FALSE;
END_IF;

IF M231 THEN
    DMOV(TRUE, 0, U3\G32);  (* Nạp Preset Value CH2 = 0 vào G32/G33 *)
    Y39 := TRUE;
    M231 := FALSE;
ELSE
    Y39 := FALSE;
END_IF;

(* 4. Đo tốc độ biến thiên xung Delta Pulse mỗi 100ms bằng phép trừ trực tiếp *)
IF SM412 THEN
    D566 := D562 - D568;
    D567 := D564 - D569;
    D568 := D562;
    D569 := D564;
END_IF;

M234 := X30; (* Module QD62D #2 Ready *)
M235 := X3A; (* Đang đếm CH1 (X3A = ON khi Y34 = ON) *)
M236 := X3B; (* Đang đếm CH2 (X3B = ON khi Y3C = ON) *)

(* ============================================================================ *)
(* 5. MODULE QX40 (SLOT 4 - 16 NGÕ VÀO DC 24V X40..X4F)                         *)
(* LƯU Ý: VÌ M LÀ HỆ THẬP PHÂN NÊN DÙNG M240..M255 (KHÔNG DÙNG CHỮ A..F)        *)
(* ============================================================================ *)
M240 := X40; M241 := X41; M242 := X42; M243 := X43;
M244 := X44; M245 := X45; M246 := X46; M247 := X47;
M248 := X48; M249 := X49; M250 := X4A; M251 := X4B;
M252 := X4C; M253 := X4D; M254 := X4E; M255 := X4F;

MOV(TRUE, K4X40, D588); (* Đọc 16 ngõ vào X40..X4F vào D588 *)

(* Bộ đếm sự kiện cạnh lên từng chân (dùng M260..M275 chốt xung) *)
IF X40 AND NOT M260 THEN D570 := D570 + 1; END_IF; M260 := X40;
IF X41 AND NOT M261 THEN D571 := D571 + 1; END_IF; M261 := X41;
IF X42 AND NOT M262 THEN D572 := D572 + 1; END_IF; M262 := X42;
IF X43 AND NOT M263 THEN D573 := D573 + 1; END_IF; M263 := X43;
IF X44 AND NOT M264 THEN D574 := D574 + 1; END_IF; M264 := X44;
IF X45 AND NOT M265 THEN D575 := D575 + 1; END_IF; M265 := X45;
IF X46 AND NOT M266 THEN D576 := D576 + 1; END_IF; M266 := X46;
IF X47 AND NOT M267 THEN D577 := D577 + 1; END_IF; M267 := X47;
IF X48 AND NOT M268 THEN D578 := D578 + 1; END_IF; M268 := X48;
IF X49 AND NOT M269 THEN D579 := D579 + 1; END_IF; M269 := X49;
IF X4A AND NOT M270 THEN D580 := D580 + 1; END_IF; M270 := X4A;
IF X4B AND NOT M271 THEN D581 := D581 + 1; END_IF; M271 := X4B;
IF X4C AND NOT M272 THEN D582 := D582 + 1; END_IF; M272 := X4C;
IF X4D AND NOT M273 THEN D583 := D583 + 1; END_IF; M273 := X4D;
IF X4E AND NOT M274 THEN D584 := D584 + 1; END_IF; M274 := X4E;
IF X4F AND NOT M275 THEN D585 := D585 + 1; END_IF; M275 := X4F;

IF M259 THEN (* Nút Reset toàn bộ bộ đếm *)
    D570 := 0; D571 := 0; D572 := 0; D573 := 0;
    D574 := 0; D575 := 0; D576 := 0; D577 := 0;
    D578 := 0; D579 := 0; D580 := 0; D581 := 0;
    D582 := 0; D583 := 0; D584 := 0; D585 := 0;
    M259 := FALSE;
END_IF;

(* ============================================================================ *)
(* 6. MODULE QY10 (SLOT 5 - 16 NGÕ RA RELAY Y50..Y5F)                           *)
(* LƯU Ý: VÌ M LÀ HỆ THẬP PHÂN NÊN DÙNG M280..M295 (KHÔNG DÙNG CHỮ A..F)        *)
(* ============================================================================ *)
IF SM402 THEN D591 := 5; END_IF;

IF M297 THEN (* Nút All ON *)
    M280 := TRUE; M281 := TRUE; M282 := TRUE; M283 := TRUE;
    M284 := TRUE; M285 := TRUE; M286 := TRUE; M287 := TRUE;
    M288 := TRUE; M289 := TRUE; M290 := TRUE; M291 := TRUE;
    M292 := TRUE; M293 := TRUE; M294 := TRUE; M295 := TRUE;
    M297 := FALSE;
END_IF;

IF M298 THEN (* Nút All OFF *)
    M280 := FALSE; M281 := FALSE; M282 := FALSE; M283 := FALSE;
    M284 := FALSE; M285 := FALSE; M286 := FALSE; M287 := FALSE;
    M288 := FALSE; M289 := FALSE; M290 := FALSE; M291 := FALSE;
    M292 := FALSE; M293 := FALSE; M294 := FALSE; M295 := FALSE;
    M298 := FALSE;
END_IF;

(* Đèn chạy tuần tự tự động (Auto Chaser nhịp 0.5s dùng xung hệ thống SM413) *)
IF M296 THEN
    IF SM413 AND NOT M299 THEN
        D590 := D590 + 1;
        IF D590 > 15 THEN D590 := 0; END_IF;
    END_IF;
    M299 := SM413;
ELSE
    D590 := 0;
    M299 := FALSE;
END_IF;


(* Xuất ngõ ra chuẩn Single-Coil: Y50..Y5F tương ứng M280..M295 *)
Y50 := (NOT M296 AND M280) OR (M296 AND (D590 = 0));
Y51 := (NOT M296 AND M281) OR (M296 AND (D590 = 1));
Y52 := (NOT M296 AND M282) OR (M296 AND (D590 = 2));
Y53 := (NOT M296 AND M283) OR (M296 AND (D590 = 3));
Y54 := (NOT M296 AND M284) OR (M296 AND (D590 = 4));
Y55 := (NOT M296 AND M285) OR (M296 AND (D590 = 5));
Y56 := (NOT M296 AND M286) OR (M296 AND (D590 = 6));
Y57 := (NOT M296 AND M287) OR (M296 AND (D590 = 7));
Y58 := (NOT M296 AND M288) OR (M296 AND (D590 = 8));
Y59 := (NOT M296 AND M289) OR (M296 AND (D590 = 9));
Y5A := (NOT M296 AND M290) OR (M296 AND (D590 = 10));
Y5B := (NOT M296 AND M291) OR (M296 AND (D590 = 11));
Y5C := (NOT M296 AND M292) OR (M296 AND (D590 = 12));
Y5D := (NOT M296 AND M293) OR (M296 AND (D590 = 13));
Y5E := (NOT M296 AND M294) OR (M296 AND (D590 = 14));
Y5F := (NOT M296 AND M295) OR (M296 AND (D590 = 15));

MOV(TRUE, K4Y50, D592); (* Ghi giá trị 16 ngõ ra Y50..Y5F vào D592 *)

(* ============================================================================ *)
(* 7. MODULE CC-LINK DAC AJ65VBTCU-68DAVN (TRẠM 1: 32 POINTS X1000..X101F)       *)
(* ============================================================================ *)
(* 1. Kiểm tra trạng thái Trạm 1 (DAC) *)
M640 := TRUE;                         (* Luôn kích hoạt xuất áp *)
M641 := X101B;                        (* Đèn báo Trạm 1 Remote READY (RX1B) *)
M642 := X101A;                        (* Đèn báo Lỗi Trạm 1 (RX1A) *)

(* 2. THIẾT LẬP THÔNG SỐ KHỞI TẠO BẮT BUỘC CHO TRẠM 1 DAC (AJ65VBTCU-68DAVN) *)
W208 := 16#0000; (* RWw8: D/A Conversion Enable cho toàn bộ CH1..CH8 (0 = ENABLE) *)
W209 := 16#0000; (* RWw9: Output Range CH1..CH4: 0H = -10V..+10V (Nạp 0..4000 = 0.0V..10.0V) *)
W20A := 16#0000; (* RWwA: Output Range CH5..CH8: 0H = -10V..+10V (Nạp 0..4000 = 0.0V..10.0V) *)
W20B := 16#0000; (* RWwB: HOLD/CLEAR Setting CH1..CH8: 0 = CLEAR về 0V khi PLC STOP *)

(* 3. NÚT RESET KHỞI TẠO LẠI (M645) HOẶC XÓA LỖI (M648) *)
IF M645 OR M648 THEN
    D670  := 0;
    M647  := FALSE; (* Cho phép chạy lại Handshake *)
    Y1018 := FALSE;
    Y1019 := FALSE;
    Y101A := TRUE;  (* Bật RY1A: Yêu cầu xóa cờ lỗi Trạm 1 *)
    IF NOT M642 THEN
        Y101A := FALSE;
        M645  := FALSE;
        M648  := FALSE;
    END_IF;
ELSE
    Y101A := FALSE;
END_IF;

(* 4. CHU TRÌNH HANDSHAKE CHUẨN XÁC THEO MANUAL MITSUBISHI SH-080397 *)
(* TỰ ĐỘNG PHỤC HỒI: Nếu module đang đòi xử lý ban đầu (X1018 ON) hoặc mất Ready (X101B OFF) *)
IF X1018 AND (D670 = 100 OR D670 = 0) THEN
    M647 := FALSE;
    D670 := 10; (* Chuyển ngay sang xử lý ban đầu theo yêu cầu của module *)
END_IF;

IF (NOT X101B) AND (D670 = 100) THEN
    M647 := FALSE;
    D670 := 0;  (* Chưa có Remote READY thì không được dừng ở bước 100 *)
END_IF;

CASE D670 OF
    0: (* Chuẩn bị bắt đầu Handshake *)
        Y1018 := FALSE;
        Y1019 := FALSE;
        D672  := 0;
        IF X1018 THEN
            D670 := 10; (* Module đòi xử lý ban đầu -> sang bước 10 *)
        ELSIF NOT X101B THEN
            D670 := 20; (* Chưa Ready -> sang bước nạp thông số *)
        ELSE
            M647 := TRUE;
            D670 := 100;
        END_IF;

    10: (* PHA 1: Initial Data Processing (Bắt tay với X1018) *)
        (* Khi module phát cờ X1018, CPU ghi RWw8..RWwB và phản hồi Y1018 = TRUE *)
        Y1018 := TRUE;
        Y1019 := FALSE;
        (* Chờ module xác nhận và tắt cờ X1018 *)
        IF NOT X1018 THEN
            Y1018 := FALSE; (* Hạ RY18 *)
            D670  := 20;    (* Sang pha nạp thông số RY19 *)
        END_IF;

    20: (* PHA 2: Initial Data Setting Request (Bật Y1019 yêu cầu module nạp Range) *)
        Y1018 := FALSE;
        Y1019 := TRUE;  (* Bật RY19: Yêu cầu module nạp dữ liệu từ RWw8..RWwB *)
        (* Chờ module nạp xong và bật cờ X1019 = TRUE *)
        IF X1019 THEN
            Y1019 := FALSE; (* Hạ RY19 *)
            D670  := 30;    (* Chờ cờ Remote READY *)
        END_IF;

    30: (* PHA 3: Chờ module hoàn tất và bật cờ X101B Remote READY *)
        Y1018 := FALSE;
        Y1019 := FALSE;
        (* Module sẽ tự tắt X1019 và bật X101B = TRUE *)
        IF (NOT X1019) AND X101B THEN
            M647  := TRUE;  (* Khởi tạo thành công 100%! *)
            D670  := 100;   (* Hoàn thành Handshake *)
        END_IF;

    100: (* TRẠNG THÁI HOẠT ĐỘNG BÌNH THƯỜNG *)
        Y1018 := FALSE;
        Y1019 := FALSE;
        M647  := X101B;     (* Duy trì cờ hoàn tất theo X101B *)
END_CASE;

(* 5. BẬT TOÀN BỘ CÁC BIT CHO PHÉP XUẤT ÁP CH1..CH8 (Y1000..Y1007) *)
Y1000 := TRUE; (* CH1 Analog Output Enable *)
Y1001 := TRUE; (* CH2 Analog Output Enable *)
Y1002 := TRUE; (* CH3 Analog Output Enable *)
Y1003 := TRUE; (* CH4 Analog Output Enable *)
Y1004 := TRUE; (* CH5 Analog Output Enable *)
Y1005 := TRUE; (* CH6 Analog Output Enable *)
Y1006 := TRUE; (* CH7 Analog Output Enable *)
Y1007 := TRUE; (* CH8 Analog Output Enable *)

(* 6. TỰ ĐỘNG NẠP MẶC ĐỊNH LÀ 10.0V (4000) ĐỂ ĐO CỰC ĐẠI THẤY NGAY *)
IF (D650 = 0) AND NOT M650 AND NOT M654 THEN
    D650 := 4000; D651 := 4000; D652 := 4000; D653 := 4000;
    D654 := 4000; D655 := 4000; D656 := 4000; D657 := 4000;
END_IF;

IF SM402 THEN
    D660 := 0; D661 := 100; M649 := FALSE;
END_IF;

(* 7. CÁC NÚT BẤM TEST XUẤT ÁP NHANH TOÀN BỘ 8 KÊNH *)
IF M650 THEN (* Set 0.0V *)
    D650 := 0; D651 := 0; D652 := 0; D653 := 0;
    D654 := 0; D655 := 0; D656 := 0; D657 := 0;
    M654 := FALSE; M650 := FALSE;
END_IF;
IF M651 THEN (* Set 2.5V *)
    D650 := 1000; D651 := 1000; D652 := 1000; D653 := 1000;
    D654 := 1000; D655 := 1000; D656 := 1000; D657 := 1000;
    M654 := FALSE; M651 := FALSE;
END_IF;
IF M652 THEN (* Set 5.0V *)
    D650 := 2000; D651 := 2000; D652 := 2000; D653 := 2000;
    D654 := 2000; D655 := 2000; D656 := 2000; D657 := 2000;
    M654 := FALSE; M652 := FALSE;
END_IF;
IF M653 THEN (* Set 10.0V *)
    D650 := 4000; D651 := 4000; D652 := 4000; D653 := 4000;
    D654 := 4000; D655 := 4000; D656 := 4000; D657 := 4000;
    M654 := FALSE; M653 := FALSE;
END_IF;

(* 8. CHẾ ĐỘ AUTO SWEEP QUÉT ĐIỆN ÁP 0V -> 10V -> 0V *)
IF M654 AND SM412 THEN
    IF NOT M649 THEN
        D660 := D660 + D661;
        IF D660 >= 4000 THEN D660 := 4000; M649 := TRUE; END_IF;
    ELSE
        D660 := D660 - D661;
        IF D660 <= 0 THEN D660 := 0; M649 := FALSE; END_IF;
    END_IF;
    D650 := D660; D651 := D660; D652 := D660; D653 := D660;
    D654 := D660; D655 := D660; D656 := D660; D657 := D660;
END_IF;

(* 9. XUẤT ÁP VÀO THANH GHI CỦA TRẠM 1 DAC (W200..W207) LIÊN TỤC *)
W200 := D650; (* CH1 Analog Value (0..4000) *)
W201 := D651; (* CH2 Analog Value *)
W202 := D652; (* CH3 Analog Value *)
W203 := D653; (* CH4 Analog Value *)
W204 := D654; (* CH5 Analog Value *)
W205 := D655; (* CH6 Analog Value *)
W206 := D656; (* CH7 Analog Value *)
W207 := D657; (* CH8 Analog Value *)

(* 10. GIÁM SÁT MÃ PHẢN HỒI VÀ TOÀN BỘ CÁC BYTE ĐẦU VÀO TỪ TRẠM 1 DAC *)
D680 := W100;      (* RWr0: Monitor CH1 Check Code *)
D681 := W108;      (* RWr8: Error Code *)
D682 := K4X1000;   (* Cờ X1000..X100F *)
D683 := K4X1010;   (* Cờ X1010..X101F (X101B = Remote READY) *)
D684 := K4X1020;   (* Cờ X1020..X102F *)
D685 := K4X1030;   (* Cờ X1030..X103F *)
D686 := W108;      (* RWr8: Error Code chuẩn theo Manual Table 3.9 *)


(* ============================================================================ *)
(* 8. MODULE CC-LINK ADC AJ65VBTCU-68ADVN (TRẠM 2: 64 POINTS X1040..X107F)       *)
(* ============================================================================ *)
(* Kiểm tra trạng thái Trạm 2 (ADC) *)
M600 := TRUE;                         (* Luôn kích hoạt đọc dữ liệu *)
M601 := X105B OR X107B;               (* Đèn báo Trạm 2 Ready *)
M602 := X105A OR X107A;               (* Đèn báo Cờ lỗi Trạm 2 *)

(* BẬT A/D CẢ 8 KÊNH TRÊN TRẠM 2 ADC (W210) *)
W210 := 16#00FF; (* Bit 0..7 = 1: Bật chuyển đổi A/D cả 8 kênh CH1..CH8 *)

IF NOT M609 THEN
    Y1059 := TRUE; Y1079 := TRUE; (* Kích cờ Initial Data Setting Request *)
    IF X1059 OR X1079 THEN        (* Trạm 2 báo đã chốt cấu hình *)
        Y1059 := FALSE; Y1079 := FALSE;
        M609  := TRUE;
    END_IF;
ELSE
    Y1059 := FALSE; Y1079 := FALSE;
END_IF;

(* Xóa lỗi & cho phép chốt lại khi nhấn nút M605 *)
IF M605 THEN
    Y105A := TRUE; Y107A := TRUE;
    M609  := FALSE;
    IF NOT M602 THEN
        Y105A := FALSE; Y107A := FALSE;
        M605  := FALSE;
    END_IF;
ELSE
    Y105A := FALSE; Y107A := FALSE;
END_IF;

(* Đọc 8 kênh Analog Input từ W110..W117 vào D600..D607 liên tục *)
D600 := W110; (* CH1 ADC Raw (0..4000) *)
D601 := W111; (* CH2 ADC Raw *)
D602 := W112; (* CH3 ADC Raw *)
D603 := W113; (* CH4 ADC Raw *)
D604 := W114; (* CH5 ADC Raw *)
D605 := W115; (* CH6 ADC Raw *)
D606 := W116; (* CH7 ADC Raw *)
D607 := W117; (* CH8 ADC Raw *)

(* Quy đổi sang mV (0..10000 mV tương ứng 0.00..10.00V) hiển thị HMI *)
D610 := (D600 * 10) / 4;
D611 := (D601 * 10) / 4;
D612 := (D602 * 10) / 4;
D613 := (D603 * 10) / 4;
D614 := (D604 * 10) / 4;
D615 := (D605 * 10) / 4;
D616 := (D606 * 10) / 4;
D617 := (D607 * 10) / 4;

IF D610 < 0 THEN D610 := 0; END_IF;
IF D611 < 0 THEN D611 := 0; END_IF;
IF D612 < 0 THEN D612 := 0; END_IF;
IF D613 < 0 THEN D613 := 0; END_IF;
IF D614 < 0 THEN D614 := 0; END_IF;
IF D615 < 0 THEN D615 := 0; END_IF;
IF D616 < 0 THEN D616 := 0; END_IF;
IF D617 < 0 THEN D617 := 0; END_IF;
END_PROGRAM

FUNCTION_BLOCK FB_TENSION_PID
VAR_INPUT
  Enable : BOOL;
  Reset : BOOL;
  Setpoint : REAL;
  Feedback : REAL;
  Kp : REAL;
  Ki : REAL;
  Kd : REAL;
  Deadband : REAL;
  Out_Min : REAL;
  Out_Max : REAL;
  AT_Enable : BOOL;
  AT_Step : REAL;
END_VAR
VAR_OUTPUT
  PID_Output : REAL;
  Error : REAL;
  AT_Done : BOOL;
  AT_Busy : BOOL;
  Tuned_Kp : REAL;
  Tuned_Ki : REAL;
  Tuned_Kd : REAL;
END_VAR
VAR
  Error_Prev : REAL;
  I_Term : REAL;
  P_Term : REAL;
  D_Term : REAL;
  AT_State : INT;
  AT_Cycle_Count : INT;
  AT_Timer_10ms : DINT;
  AT_Period_Tu : REAL;
  AT_Ku : REAL;
  AT_PV_Max : REAL;
  AT_PV_Min : REAL;
  AT_Base_Out : REAL;
  AT_Relay_State : BOOL;
  Test_Step : REAL;
END_VAR
(* ============================================================================ *)
(* FUNCTION BLOCK: FB_TENSION_PID (ĐIỀU KHIỂN PID & AUTO-TUNING TỰ ĐỘNG TÌM THÔNG SỐ) *)
(* PHƯƠNG PHÁP AUTO-TUNING: RELAY FEEDBACK LIMIT-CYCLE (ZIEGLER-NICHOLS CẢI TIẾN) *)
(* ============================================================================ *)

IF NOT Enable THEN
    PID_Output := 0.0;
    I_Term     := 0.0;
    Error_Prev := 0.0;
    AT_Busy    := FALSE;
    AT_State   := 0;
    RETURN;
END_IF;

IF Reset THEN
    I_Term     := 0.0;
    Error_Prev := 0.0;
    PID_Output := 0.0;
    AT_Busy    := FALSE;
    AT_State   := 0;
    AT_Done    := FALSE;
    RETURN;
END_IF;

(* ============================================================================ *)
(* 1. CHẾ ĐỘ AUTO-TUNING (DÒ THÔNG SỐ TỰ ĐỘNG BẰNG RELAY LIMIT-CYCLE)           *)
(* ============================================================================ *)
IF AT_Enable THEN
    AT_Busy := TRUE;
    AT_Done := FALSE;
    
    (* Sử dụng biến nội bộ Test_Step để không ghi đè vào VAR_INPUT AT_Step *)
    IF AT_Step > 0.0 THEN
        Test_Step := AT_Step;
    ELSE
        Test_Step := 800.0; (* Mặc định 800 đơn vị DAC ~ 5% của 16000 *)
    END_IF;

    CASE AT_State OF
        0: (* KHỞI TẠO BƯỚC TEST *)
            AT_Base_Out     := PID_Output;
            AT_PV_Max       := Feedback;
            AT_PV_Min       := Feedback;
            AT_Cycle_Count  := 0;
            AT_Timer_10ms   := 0;
            AT_Relay_State  := TRUE;
            AT_State        := 1;

        1: (* THỰC THI DAO ĐỘNG BẬT/TẮT RELAY QUA SETPOINT *)
            AT_Timer_10ms := AT_Timer_10ms + 1;

            (* Theo dõi giá trị đỉnh/đáy của Feedback *)
            IF Feedback > AT_PV_Max THEN AT_PV_Max := Feedback; END_IF;
            IF Feedback < AT_PV_Min THEN AT_PV_Min := Feedback; END_IF;

            (* Điều khiển Relay đảo trạng thái khi vượt qua Setpoint *)
            IF AT_Relay_State THEN
                PID_Output := AT_Base_Out + Test_Step;
                IF Feedback >= Setpoint THEN
                    AT_Relay_State := FALSE;
                END_IF;
            ELSE
                PID_Output := AT_Base_Out - Test_Step;
                IF Feedback < Setpoint THEN
                    AT_Relay_State := TRUE;
                    AT_Cycle_Count := AT_Cycle_Count + 1; (* Đếm xong 1 chu kỳ hoàn chỉnh *)
                END_IF;
            END_IF;

            (* Khi hoàn thành đủ 3 chu kỳ dao động chuẩn *)
            IF AT_Cycle_Count >= 3 THEN
                AT_State := 2;
            END_IF;

        2: (* TÍNH TOÁN BỘ THÔNG SỐ TUNED_KP, TUNED_KI, TUNED_KD *)
            (* Chu kỳ dao động riêng Tu (giây) = tổng thời gian 3 chu kỳ / 3 *)
            IF AT_Timer_10ms > 0 THEN
                AT_Period_Tu := (DINT_TO_REAL(AT_Timer_10ms) * 0.01) / 3.0;
            ELSE
                AT_Period_Tu := 1.0;
            END_IF;

            (* Biên độ dao động đáp ứng A = (PV_Max - PV_Min) / 2 *)
            IF (AT_PV_Max - AT_PV_Min) > 0.1 THEN
                (* Độ khuếch đại tới hạn Ku = 4 * Test_Step / (PI * A) *)
                AT_Ku := (4.0 * Test_Step) / (3.141593 * ((AT_PV_Max - AT_PV_Min) / 2.0));
            ELSE
                AT_Ku := 1.0;
            END_IF;

            (* TÍNH THEO CÔNG THỨC ZIEGLER-NICHOLS CHỐNG VỌT LỐ (NO-OVERSHOOT) *)
            Tuned_Kp := AT_Ku * 0.35;                   (* Kp an toàn êm ái *)
            
            IF AT_Period_Tu > 0.05 THEN
                Tuned_Ki := Tuned_Kp * (0.01 / (AT_Period_Tu * 0.85)); (* Ki cho chu kỳ 10ms *)
                Tuned_Kd := Tuned_Kp * ((AT_Period_Tu * 0.12) / 0.01); (* Kd cho chu kỳ 10ms *)
            ELSE
                Tuned_Ki := Tuned_Kp * 0.05;
                Tuned_Kd := Tuned_Kp * 0.02;
            END_IF;

            (* Khống chế biên an toàn *)
            IF Tuned_Kp < 0.1 THEN Tuned_Kp := 0.1; ELSIF Tuned_Kp > 20.0 THEN Tuned_Kp := 20.0; END_IF;
            IF Tuned_Ki < 0.001 THEN Tuned_Ki := 0.001; ELSIF Tuned_Ki > 5.0 THEN Tuned_Ki := 5.0; END_IF;
            IF Tuned_Kd < 0.0 THEN Tuned_Kd := 0.0; ELSIF Tuned_Kd > 5.0 THEN Tuned_Kd := 5.0; END_IF;

            AT_Busy  := FALSE;
            AT_Done  := TRUE;
            AT_State := 0;
    END_CASE;

    (* Giới hạn biên đầu ra trong lúc test *)
    IF PID_Output > Out_Max THEN PID_Output := Out_Max; END_IF;
    IF PID_Output < Out_Min THEN PID_Output := Out_Min; END_IF;
    RETURN;
END_IF;

(* Khi tắt AT_Enable *)
IF AT_Busy THEN
    AT_Busy  := FALSE;
    AT_State := 0;
END_IF;

(* ============================================================================ *)
(* 2. CHẾ ĐỘ ĐIỀU KHIỂN PID TIÊU CHUẨN (NORMAL RUNNING)                        *)
(* ============================================================================ *)

(* 1. TÍNH ĐỘ LỆCH ERROR E(K) *)
Error := Setpoint - Feedback;

(* 2. BỘ LỌC VÙNG CHẾT DEADBAND *)
IF ABS(Error) <= Deadband THEN
    Error := 0.0;
END_IF;

(* 3. TÍNH THÀNH PHẦN PROPORTIONAL (P) *)
P_Term := Error * Kp;

(* 4. TÍNH THÀNH PHẦN INTEGRAL (I) VỚI CHỐNG BÃO HÒA ANTI-WINDUP *)
I_Term := I_Term + (Error * Ki);

IF Out_Max > Out_Min THEN
    IF I_Term > Out_Max THEN
        I_Term := Out_Max;
    ELSIF I_Term < Out_Min THEN
        I_Term := Out_Min;
    END_IF;
END_IF;

(* 5. TÍNH THÀNH PHẦN DERIVATIVE (D) *)
D_Term := (Error - Error_Prev) * Kd;
Error_Prev := Error;

(* 6. TỔNG HỢP NỔI PID VÀ ÉP BIÊN OUT_MIN..OUT_MAX *)
PID_Output := P_Term + I_Term + D_Term;

IF Out_Max > Out_Min THEN
    IF PID_Output > Out_Max THEN
        PID_Output := Out_Max;
    ELSIF PID_Output < Out_Min THEN
        PID_Output := Out_Min;
    END_IF;
END_IF;
END_FUNCTION_BLOCK

PROGRAM POU_INIT
(* ============================================================================ *)
(* TÊN CHƯƠNG TRÌNH : INIT_PROGRAM (INITIAL EXECUTION POU - KHỞI TẠO HỆ THỐNG)    *)
(* HỆ THỐNG        : MÁY GHÉP MÀNG METALIZE TỰ ĐỘNG - MITSUBISHI Q02U PLC       *)
(* KIỂU DỮ LIỆU    : SỐ THỰC FLOAT / REAL (CHUẨN IEC)                          *)
(* CẤU TRÚC PHẦN CỨNG MỚI (DIRECT BASE RACK - KHÔNG DÙNG CC-LINK):             *)
(*   - SLOT 0 (H00): Q68ADV (8 CH Analog Input: Loadcell T, X1, M, U & Analog S)*)
(*   - SLOT 1 (H10): Q68DAV (8 CH Analog Output: Speed/Torque T, X1, X2, Ms, S, M, U) *)
(*   - SLOT 2 (H20): QD62D  (2 CH High Speed Counter: Trục T & Trục X1)        *)
(*   - SLOT 3 (H30): QD62D  (2 CH High Speed Counter: Trục X2 & Trục Ms)       *)
(*   - SLOT 4 (H40): QX40   (16 CH Digital Input: X40..X4F)                    *)
(*   - SLOT 5 (H50): QY40   (16 CH Digital Output: Y50..Y5F)                   *)
(*   - SLOT 6 (H60): QJ71C24N (RS232/RS485 Communication)                      *)
(* ============================================================================ *)

(* ---------------------------------------------------------------------------- *)
(* 1. KHỞI TẠO TỐC ĐỘ TỐI ĐA MOTOR (RPM - REAL)                                *)
(* ---------------------------------------------------------------------------- *)
IF Max_RPM_X2 <= 0.0 THEN Max_RPM_X2 := 1000.0; END_IF; (* Trục Master X2: Max 1000 RPM *)
IF Max_RPM_X1 <= 0.0 THEN Max_RPM_X1 := 1000.0; END_IF; (* Trục Kéo X1:    Max 1000 RPM *)
IF Max_RPM_Ms <= 0.0 THEN Max_RPM_Ms := 3000.0; END_IF; (* Trục Ghép Ms:   Max 3000 RPM *)
IF Max_RPM_S  <= 0.0 THEN Max_RPM_S  := 3000.0; END_IF; (* Trục Dầu S:     Max 3000 RPM *)
IF Max_RPM_T  <= 0.0 THEN Max_RPM_T  := 1500.0; END_IF; (* Trục Thu T:     Max 1500 RPM *)

(* ---------------------------------------------------------------------------- *)
(* 2. KHỞI TẠO TỶ SỐ TRUYỀN HỘP SỐ THỰC TẾ (GEAR RATIO - REAL)                *)
(* ---------------------------------------------------------------------------- *)
IF Gear_Ratio_T  <= 0.0 THEN Gear_Ratio_T  := 10.1; END_IF; (* Thu T:     10.1 : 1 (D620) *)
IF Gear_Ratio_X1 <= 0.0 THEN Gear_Ratio_X1 := 8.0;  END_IF; (* Xả X1:     8.0  : 1 (D622) *)
IF Gear_Ratio_X2 <= 0.0 THEN Gear_Ratio_X2 := 8.0;  END_IF; (* Master X2: 8.0  : 1 (D624) *)
IF Gear_Ratio_Ms <= 0.0 THEN Gear_Ratio_Ms := 10.0; END_IF; (* Ghép Ms:   10.0 : 1 (D626) *)
IF Gear_Ratio_S  <= 0.0 THEN Gear_Ratio_S  := 10.0; END_IF; (* Dầu S:     10.0 : 1 (D628) *)
IF Gear_Ratio_U  <= 0.0 THEN Gear_Ratio_U  := 1.03125; END_IF; (* Trục Xả Metalize U: Gear = 33/32 = 1.03125 (D210) *)

(* ---------------------------------------------------------------------------- *)
(* 3. KHỞI TẠO ĐƯỜNG KÍNH LÔ CƠ CẤU (ROLLER DIAMETER - mm - REAL)              *)
(* ---------------------------------------------------------------------------- *)
IF Dia_X1_Roller_mm <= 0.0 THEN Dia_X1_Roller_mm := 300.5; END_IF; (* Lô Kéo X1:    300.5 mm (D638) *)
IF Dia_X2_Roller_mm <= 0.0 THEN Dia_X2_Roller_mm := 300.5; END_IF; (* Lô Master X2: 300.5 mm (D642) *)
IF Dia_Ms_Roller_mm <= 0.0 THEN Dia_Ms_Roller_mm := 200.0; END_IF; (* Lô Ghép Ms:   200.0 mm (D640) *)
IF Dia_S_Roller_mm  <= 0.0 THEN Dia_S_Roller_mm  := 100.0; END_IF; (* Lô Dầu S:     100.0 mm (D648) *)

(* ---------------------------------------------------------------------------- *)
(* 4. KHỞI TẠO ĐƯỜNG KÍNH LÕI (CORE) VÀ ĐƯỜNG KÍNH MAX (MAX DIA) (mm - REAL)    *)
(* ---------------------------------------------------------------------------- *)
IF Core_Dia_T_mm <= 0.0 THEN Core_Dia_T_mm := 76.0;   END_IF; (* Lõi cuộn Thu T:  76.0 mm (D644) *)
IF Core_Dia_M_mm <= 0.0 THEN Core_Dia_M_mm := 76.0;   END_IF; (* Lõi cuộn Xả M:   76.0 mm (D645) *)
IF Core_Dia_U_mm <= 0.0 THEN Core_Dia_U_mm := 76.0;   END_IF; (* Lõi cuộn Xả U:   76.0 mm (D647) *)

IF Max_Dia_T_mm  <= 0.0 THEN Max_Dia_T_mm  := 1000.0; END_IF; (* Cuộn Thu T max: 1000.0 mm (D646) *)
IF Max_Dia_M_mm  <= 0.0 THEN Max_Dia_M_mm  := 600.0;  END_IF; (* Cuộn Xả M max:   600.0 mm (D649) *)
IF Max_Dia_U_mm  <= 0.0 THEN Max_Dia_U_mm  := 800.0;  END_IF; (* Cuộn Xả U max:   800.0 mm (D650) *)

(* ---------------------------------------------------------------------------- *)
(* 5. KHỞI TẠO ĐƯỜNG KÍNH BAN ĐẦU KHI MỚI BẬT NGUỒN (REAL)                     *)
(* ---------------------------------------------------------------------------- *)
IF Real_Dia_T_mm < Core_Dia_T_mm OR Real_Dia_T_mm > Max_Dia_T_mm THEN
    Real_Dia_T_mm := Core_Dia_T_mm; (* 76.0 mm - D724 *)
END_IF;

IF Real_Dia_M_mm < Core_Dia_M_mm OR Real_Dia_M_mm > Max_Dia_M_mm THEN
    Real_Dia_M_mm := Max_Dia_M_mm;  (* 600.0 mm - D722 *)
END_IF;

IF Real_Dia_U_mm < Core_Dia_U_mm OR Real_Dia_U_mm > Max_Dia_U_mm THEN
    Real_Dia_U_mm := Max_Dia_U_mm;  (* 800.0 mm - D720 *)
END_IF;

(* ---------------------------------------------------------------------------- *)
(* 6. KHỞI TẠO TỶ LỆ TỐC ĐỘ VÀ BÙ TỐC (SPEED RATIO - REAL, 1.0 = 100%)         *)
(* ---------------------------------------------------------------------------- *)
IF Speed_Ratio_T  <= 0.0 THEN Speed_Ratio_T  := 1.05; END_IF; (* Chạy nhanh hơn 5% giữ căng (D756) *)
IF Speed_Ratio_X1 <= 0.0 THEN Speed_Ratio_X1 := 1.00; END_IF; (* Đồng bộ 100.0% (D758) *)
IF Speed_Ratio_Ms <= 0.0 THEN Speed_Ratio_Ms := 1.00; END_IF; (* Đồng bộ 100.0% (D762) *)
IF Speed_Ratio_S  <= 0.0 THEN Speed_Ratio_S  := 1.00; END_IF; (* Đồng bộ 100.0% (D766) *)

(* ---------------------------------------------------------------------------- *)
(* 7. KHỞI TẠO GIỚI HẠN TỐC ĐỘ DÂY CHUYỀN (m/phút - REAL)                      *)
(* ---------------------------------------------------------------------------- *)
IF Max_Speed_MPM         <= 0.0 THEN Max_Speed_MPM         := 100.0; END_IF; (* Max 100.0 m/p (D602) *)
IF Min_Speed_MPM         <= 0.0 THEN Min_Speed_MPM         := 2.0;   END_IF; (* Min 2.0 m/p (D603) *)
IF Release_Pen_Speed_MPM <= 0.0 THEN Release_Pen_Speed_MPM := 2.0;   END_IF; (* Tốc độ nhả pen (D604) *)
IF Ramp_Accel_Rate       <= 0.0 THEN Ramp_Accel_Rate       := 0.5;   END_IF; (* Gia tốc tăng tốc (D606) *)
IF Ramp_Decel_Rate       <= 0.0 THEN Ramp_Decel_Rate       := 1.0;   END_IF; (* Gia tốc giảm tốc (D608) *)
IF Decel_Distance_Meters <= 0.0 THEN Decel_Distance_Meters := 50.0;  END_IF; (* Khoảng cách hãm dừng (m) *)

(* ---------------------------------------------------------------------------- *)
(* 8. KHỞI TẠO CÀI ĐẶT LỰC CĂNG (TENSION SP - kg/N - REAL) & HỆ SỐ PID         *)
(* ---------------------------------------------------------------------------- *)
IF SP_Tension_T  <= 0.0 THEN SP_Tension_T  := 15.0; END_IF; (* SP Lực căng Thu T: 15.0 kg (D660) *)
IF SP_Tension_X1 <= 0.0 THEN SP_Tension_X1 := 12.0; END_IF; (* SP Lực căng Xả X1: 12.0 kg (D662) *)
IF SP_Tension_M  <= 0.0 THEN SP_Tension_M  := 10.0; END_IF; (* SP Lực căng Xả M:  10.0 kg (D664) *)
IF SP_Tension_U  <= 0.0 THEN SP_Tension_U  := 10.0; END_IF; (* SP Lực căng Xả U:  10.0 kg (D668) *)

(* Hệ số PID cuộn Thu T *)
IF Kp_T <= 0.0 THEN Kp_T := 1.5; END_IF;
IF Ki_T <= 0.0 THEN Ki_T := 0.2; END_IF;
IF Kd_T <= 0.0 THEN Kd_T := 0.1; END_IF;

(* Hệ số PID cuộn Xả X1 *)
IF Kp_X1 <= 0.0 THEN Kp_X1 := 1.2; END_IF;
IF Ki_X1 <= 0.0 THEN Ki_X1 := 0.15; END_IF;
IF Kd_X1 <= 0.0 THEN Kd_X1 := 0.08; END_IF;

(* Hệ số PID trục Master X2 *)
IF Kp_X2 <= 0.0 THEN Kp_X2 := 1.0; END_IF;
IF Ki_X2 <= 0.0 THEN Ki_X2 := 0.1; END_IF;
IF Kd_X2 <= 0.0 THEN Kd_X2 := 0.05; END_IF;

(* Hệ số PID trục Ghép Ms *)
IF Kp_Ms <= 0.0 THEN Kp_Ms := 1.0; END_IF;
IF Ki_Ms <= 0.0 THEN Ki_Ms := 0.1; END_IF;
IF Kd_Ms <= 0.0 THEN Kd_Ms := 0.05; END_IF;

(* Hệ số PID trục Dầu S *)
IF Kp_S <= 0.0 THEN Kp_S := 1.0; END_IF;
IF Ki_S <= 0.0 THEN Ki_S := 0.1; END_IF;
IF Kd_S <= 0.0 THEN Kd_S := 0.05; END_IF;

(* Hệ số PID cuộn Thắng M *)
IF Kp_M <= 0.0 THEN Kp_M := 1.0; END_IF;
IF Ki_M <= 0.0 THEN Ki_M := 0.1; END_IF;
IF Kd_M <= 0.0 THEN Kd_M := 0.05; END_IF;

(* Hệ số PID cuộn Xả U *)
IF Kp_U <= 0.0 THEN Kp_U := 1.0; END_IF;
IF Ki_U <= 0.0 THEN Ki_U := 0.1; END_IF;
IF Kd_U <= 0.0 THEN Kd_U := 0.05; END_IF;

(* ---------------------------------------------------------------------------- *)
(* 9. KHỞI TẠO TORQUE HÃM MIN / MAX VÀ GIỮ DỪNG MÁY (% - REAL)                 *)
(* ---------------------------------------------------------------------------- *)
IF Min_Torque_M          <= 0.0 THEN Min_Torque_M          := 4.0;  END_IF; (* 4.0 % *)
IF Max_Torque_M          <= 0.0 THEN Max_Torque_M          := 20.0; END_IF; (* 20.0 % *)
IF Init_Holding_Torque_M <= 0.0 THEN Init_Holding_Torque_M := 8.0;  END_IF; (* 8.0 % *)

IF Min_Torque_U          <= 0.0 THEN Min_Torque_U          := 5.0;  END_IF; (* 5.0 % *)
IF Max_Torque_U          <= 0.0 THEN Max_Torque_U          := 25.0; END_IF; (* 25.0 % *)
IF Init_Holding_Torque_U <= 0.0 THEN Init_Holding_Torque_U := 10.0; END_IF; (* 10.0 % *)

(* ---------------------------------------------------------------------------- *)
(* 10. KHỞI TẠO HỆ SỐ GAIN CALIB LOADCELL (REAL)                                *)
(* ---------------------------------------------------------------------------- *)
IF Calib_Gain_T  <= 0.0 THEN Calib_Gain_T  := 1.0; END_IF;
IF Calib_Gain_X1 <= 0.0 THEN Calib_Gain_X1 := 1.0; END_IF;
IF Calib_Gain_M  <= 0.0 THEN Calib_Gain_M  := 1.0; END_IF;
IF Calib_Gain_U  <= 0.0 THEN Calib_Gain_U  := 1.0; END_IF;

(* ---------------------------------------------------------------------------- *)
(* 11. KHỞI TẠO CẤU HÌNH MODULE Q68ADV (SLOT 0 - HEAD ADDRESS H00)             *)
(* ---------------------------------------------------------------------------- *)
(* BFM #0: Cho phép chuyển đổi A/D cả 8 kênh (0 = Enable, 1 = Disable)          *)
U0\G0 := 16#0000; (* Enable toàn bộ CH1..CH8 *)

(* BFM #9 & #10: Cài đặt chế độ lọc trung bình trượt (Moving Average = 16#3333) *)
U0\G9  := 16#3333; (* CH1..CH4: Moving Average *)
U0\G10 := 16#3333; (* CH5..CH8: Moving Average *)

(* BFM #11..#18: Số lượng mẫu trung bình trượt (16 mẫu liên tục)                *)
U0\G11 := 16; (* CH1: Loadcell Thu T *)
U0\G12 := 16; (* CH2: Loadcell Kéo X1 *)
U0\G13 := 16; (* CH3: Loadcell Thắng M *)
U0\G14 := 16; (* CH4: Loadcell Xả U *)
U0\G15 := 16; (* CH5: Analog Tốc độ Servo Trục S *)
U0\G16 := 16; (* CH6: Dự phòng *)
U0\G17 := 16; (* CH7: Dự phòng *)
U0\G18 := 16; (* CH8: Dự phòng *)

(* ---------------------------------------------------------------------------- *)
(* 12. KHỞI TẠO CẤU HÌNH MODULE Q68DAV (SLOT 1 - HEAD ADDRESS H10)             *)
(* ---------------------------------------------------------------------------- *)
(* BFM #0: Cho phép chuyển đổi D/A cả 8 kênh (0 = Enable, 1 = Disable)          *)
U1\G0 := 16#0000; (* Enable D/A cho CH1..CH8 *)

(* BFM #9: Cho phép ngõ ra Analog Output (Bit 0..7: 1 = Output Enable)          *)
U1\G9 := 16#00FF; (* Cho phép xuất áp ra cả 8 kênh *)

(* Bật cờ Y11 hoặc Y10 cho phép chuyển đổi D/A *)
Y11 := TRUE;
END_PROGRAM

// device comments not shown above
D524  ; DAC CH1: Speed Thu T
D526  ; DAC CH3: Speed Xa X1
D530  ; DAC CH7: Speed Trang Dau S
D531  ; DAC CH8: Speed Xa U
X50  ; "X","50","Sensor tiem can dem vo
X51  ; "X","51","Sensor tiem can dem vo
SM402  ; After RUN, ON for 1 scan only
SM409  ; 0.01 second clock
SM412  ; 1 second clock
SM413  ; 2 second clock
M1104  ; Remote Input X0 (St4)
M1105  ; Remote Input X1 (St4)
M1106  ; Remote Input X2 (St4)
M1107  ; Remote Input X3 (St4)
M1108  ; Remote Input X4 (St4)
M1109  ; Remote Input X5 (St4)
M1110  ; Remote Input X6 (St4)
M1111  ; Remote Input X7 (St4)
M1208  ; Cho phép chuyển đổi A/D Trạm 1 (
M1240  ; Cho phép chuyển đổi D/A Trạm 2 (
M1304  ; Servo ON Truc Thu T (Y8)
M1305  ; Servo ON Truc Xa X1 (Y9)
M1306  ; Servo ON Truc Master X2 (YA)
M1307  ; Servo ON Truc Ghep Ms (YB)
M1308  ; Servo ON Truc Trang Dau S (YC)
M1309  ; Solenoid Valve Pen 1 (YD)
M1310  ; Solenoid Valve Pen 2 (YE)
M1311  ; Du phong / Bao loi (YF)
D525  ; DAC CH2: Torque Thu T
D527  ; DAC CH4: Speed Master X2
D528  ; DAC CH5: Speed Ghep Ms
D529  ; DAC CH6: Torque Ghep Ms
X52  ; "X","52","Nut nhan START vat ly
X53  ; "X","53","Nut nhan STOP vat ly (
X54  ; "X","54","Nut nhan INC Tang toc
X55  ; "X","55","Nut nhan DEC Giam toc
X56  ; "X","56","Nut Toggle Pen 1 vat l
X57  ; "X","57","Nut Toggle Pen 2 vat l
X58  ; "X","58","Cong tac Giu Torque M
X59  ; "X","59","Cong tac Giu Torque U
X5A  ; "X","5A","Cong tac Rua may bo ch
X5B  ; "X","5B","Cong tac Rua may bo ch
X5C  ; "X","5C","Nut nhan co BO CHAM NO
